SUBAPPLICATION ACTION_CLIENT
  (* Standard: 61499-2 *)
  (* Version 1.0, 2023-03-21, Tim Hesse *)
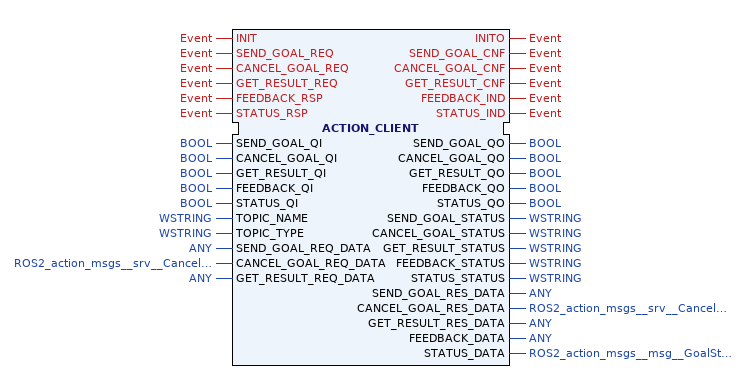
  EVENT_INPUT
    INIT; (* Initialization Request *)
    SEND_GOAL_REQ; (* Send Goal Request *)
    CANCEL_GOAL_REQ; (* Cancel Goal Request *)
    GET_RESULT_REQ; (* Get Result Request *)
    FEEDBACK_RSP; (* Application Response to FEEDBACK_IND *)
    STATUS_RSP;
  END_EVENT
  EVENT_OUTPUT
    INITO; (* Initialization Confirm *)
    SEND_GOAL_CNF; (* Send Goal Confirmation *)
    CANCEL_GOAL_CNF; (* Cancel Goal Confirmation *)
    GET_RESULT_CNF; (* Get Result Confirmation *)
    FEEDBACK_IND; (* Confirmation of Feedback *)
    STATUS_IND;
  END_EVENT
  VAR_INPUT
    SEND_GOAL_QI : BOOL; (* Send Goal Input Event Qualifier *)
    CANCEL_GOAL_QI : BOOL; (* Cancel Goal Input Event Qualifier *)
    GET_RESULT_QI : BOOL; (* Get Result Input Event Qualifier *)
    FEEDBACK_QI : BOOL; (* Feedback Input Event Qualifier *)
    STATUS_QI : BOOL;
    TOPIC_NAME : WSTRING; (* ROS 2 Topic Name *)
    TOPIC_TYPE : WSTRING; (* ROS 2 Topic Type *)
    SEND_GOAL_REQ_DATA : ANY; (* Send Goal Request Data *)
    CANCEL_GOAL_REQ_DATA : ROS2_action_msgs__srv__CancelGoal__Request; (* Cancel Goal Request Data *)
    GET_RESULT_REQ_DATA : ANY; (* Get Result Request Data *)
  END_VAR
  VAR_OUTPUT
    SEND_GOAL_QO : BOOL; (* Send Goal Output Event Qualifier *)
    CANCEL_GOAL_QO : BOOL; (* Cancel Goal Output Event Qualifier *)
    GET_RESULT_QO : BOOL; (* Get Result Output Event Qualifier *)
    FEEDBACK_QO : BOOL; (* Feedback Output Event Qualifier *)
    STATUS_QO : BOOL;
    SEND_GOAL_STATUS : WSTRING; (* Send Goal Service Status *)
    CANCEL_GOAL_STATUS : WSTRING; (* Cancel Goal Service Status *)
    GET_RESULT_STATUS : WSTRING; (* Get Result Service Status *)
    FEEDBACK_STATUS : WSTRING; (* Feedback Subscriber Status *)
    STATUS_STATUS : WSTRING;
    SEND_GOAL_RES_DATA : ANY; (* Send Goal Response Data *)
    CANCEL_GOAL_RES_DATA : ROS2_action_msgs__srv__CancelGoal__Response; (* Cacnel Goal Response Data *)
    GET_RESULT_RES_DATA : ANY; (* Get Result Response Data *)
    FEEDBACK_DATA : ANY; (* Feedback Data *)
    STATUS_DATA : ROS2_action_msgs__msg__GoalStatusArray;
  END_VAR
  FBS
    E_REND : E_REND;
    E_REND_1 : E_REND;
    E_REND_2 : E_REND;
    E_REND_3 : E_REND;
  END_FBS
  SUBAPPS
    ACTION_CLIENT_SEND_GOAL : ACTION_CLIENT_SEND_GOAL;
    ACTION_CLIENT_CANCEL_GOAL : ACTION_CLIENT_CANCEL_GOAL;
    ACTION_CLIENT_GET_RESULT : ACTION_CLIENT_GET_RESULT;
    ACTION_CLIENT_FEEDBACK_MESSAGE : ACTION_CLIENT_FEEDBACK_MESSAGE;
    ACTION_CLIENT_STATUS : ACTION_CLIENT_STATUS;
  END_SUBAPPS
  EVENT_CONNECTIONS
    SEND_GOAL_REQ TO ACTION_CLIENT_SEND_GOAL.REQ;
    CANCEL_GOAL_REQ TO ACTION_CLIENT_CANCEL_GOAL.REQ;
    GET_RESULT_REQ TO ACTION_CLIENT_GET_RESULT.REQ;
    FEEDBACK_RSP TO ACTION_CLIENT_FEEDBACK_MESSAGE.RSP;
    ACTION_CLIENT_SEND_GOAL.CNF TO SEND_GOAL_CNF;
    ACTION_CLIENT_CANCEL_GOAL.CNF TO CANCEL_GOAL_CNF;
    ACTION_CLIENT_GET_RESULT.CNF TO GET_RESULT_CNF;
    ACTION_CLIENT_FEEDBACK_MESSAGE.IND TO FEEDBACK_IND;
    STATUS_RSP TO ACTION_CLIENT_STATUS.RSP;
    ACTION_CLIENT_STATUS.IND TO STATUS_IND;
    E_REND.EO TO E_REND_2.EI1;
    E_REND_1.EO TO E_REND_2.EI2;
    ACTION_CLIENT_SEND_GOAL.INITO TO E_REND.EI1;
    ACTION_CLIENT_CANCEL_GOAL.INITO TO E_REND.EI2;
    ACTION_CLIENT_GET_RESULT.INITO TO E_REND_1.EI1;
    ACTION_CLIENT_FEEDBACK_MESSAGE.INITO TO E_REND_1.EI2;
    E_REND_2.EO TO E_REND_3.EI2;
    E_REND_3.EO TO INITO;
    ACTION_CLIENT_STATUS.INITO TO E_REND_3.EI1;
    INIT TO ACTION_CLIENT_SEND_GOAL.INIT;
    INIT TO ACTION_CLIENT_GET_RESULT.INIT;
    INIT TO ACTION_CLIENT_CANCEL_GOAL.INIT;
    INIT TO ACTION_CLIENT_FEEDBACK_MESSAGE.INIT;
    INIT TO ACTION_CLIENT_STATUS.INIT;
  END_CONNECTIONS
  DATA_CONNECTIONS
    SEND_GOAL_QI TO ACTION_CLIENT_SEND_GOAL.QI;
    SEND_GOAL_REQ_DATA TO ACTION_CLIENT_SEND_GOAL.REQ_DATA;
    CANCEL_GOAL_QI TO ACTION_CLIENT_CANCEL_GOAL.QI;
    CANCEL_GOAL_REQ_DATA TO ACTION_CLIENT_CANCEL_GOAL.REQ_DATA;
    GET_RESULT_QI TO ACTION_CLIENT_GET_RESULT.QI;
    GET_RESULT_REQ_DATA TO ACTION_CLIENT_GET_RESULT.REQ_DATA;
    FEEDBACK_QI TO ACTION_CLIENT_FEEDBACK_MESSAGE.QI;
    ACTION_CLIENT_SEND_GOAL.QO TO SEND_GOAL_QO;
    ACTION_CLIENT_SEND_GOAL.STATUS TO SEND_GOAL_STATUS;
    ACTION_CLIENT_SEND_GOAL.RES_DATA TO SEND_GOAL_RES_DATA;
    ACTION_CLIENT_CANCEL_GOAL.QO TO CANCEL_GOAL_QO;
    ACTION_CLIENT_CANCEL_GOAL.STATUS TO CANCEL_GOAL_STATUS;
    ACTION_CLIENT_CANCEL_GOAL.RES_DATA TO CANCEL_GOAL_RES_DATA;
    ACTION_CLIENT_GET_RESULT.QO TO GET_RESULT_QO;
    ACTION_CLIENT_GET_RESULT.STATUS TO GET_RESULT_STATUS;
    ACTION_CLIENT_GET_RESULT.RES_DATA TO GET_RESULT_RES_DATA;
    ACTION_CLIENT_FEEDBACK_MESSAGE.QO TO FEEDBACK_QO;
    ACTION_CLIENT_FEEDBACK_MESSAGE.STATUS TO FEEDBACK_STATUS;
    ACTION_CLIENT_FEEDBACK_MESSAGE.SUB_DATA TO FEEDBACK_DATA;
    STATUS_QI TO ACTION_CLIENT_STATUS.QI;
    ACTION_CLIENT_STATUS.STATUS TO STATUS_STATUS;
    ACTION_CLIENT_STATUS.SUB_DATA TO STATUS_DATA;
    ACTION_CLIENT_STATUS.QO TO STATUS_QO;
    TOPIC_NAME TO ACTION_CLIENT_SEND_GOAL.TOPIC_NAME;
    TOPIC_TYPE TO ACTION_CLIENT_SEND_GOAL.TOPIC_TYPE;
    TOPIC_NAME TO ACTION_CLIENT_CANCEL_GOAL.TOPIC_NAME;
    TOPIC_NAME TO ACTION_CLIENT_GET_RESULT.TOPIC_NAME;
    TOPIC_TYPE TO ACTION_CLIENT_GET_RESULT.TOPIC_TYPE;
    TOPIC_NAME TO ACTION_CLIENT_FEEDBACK_MESSAGE.TOPIC_NAME;
    TOPIC_TYPE TO ACTION_CLIENT_FEEDBACK_MESSAGE.TOPIC_TYPE;
    TOPIC_NAME TO ACTION_CLIENT_STATUS.TOPIC_NAME;
  END_CONNECTIONS
END_SUBAPPLICATION
